// TIA Portal V16 export
// export: Created 2024-09-05T17:36:33.8079736Z, ExportSetting WithDefaults, DisplayName Totally Integrated Automation Portal, DisplayVersion V16 Update 6, DisplayName TIA Portal Version Control Interface, DisplayVersion V16 Update 2, DisplayName TIA Portal Openness, DisplayVersion V16 Update 6, DisplayName STEP 7 Professional, DisplayVersion V16 Update 6, DisplayName STEP 7 Safety, DisplayVersion V16, DisplayName WinCC Advanced, DisplayVersion V16 Update 6
VAR_GLOBAL   // PLC tag table "Modes"
END_VAR
VAR_GLOBAL CONSTANT   // user constants
   mode_0_not_selected : Int := 0;
   mode_3_automat : Int := 3;
   mode_2_base : Int := 2;
   mode_1_manual : Int := 1;
   mode_4_semiautomat : Int := 4;
END_VAR
